// TIA Portal V20 export
TYPE "LKinCtrl_typePointParameter_reduced"
   STRUCT
      pathDynamics : "LKinCtrl_typePathDynamics";   // dynamics settings for single command
      orientationDirection : DInt := 3;   // 1: positive direction; 2: negative direction; 3: shortest distance
      bufferMode : DInt := 1;   // 1: standstill between commands, 2: blending with lower speed; 5: blending with higher speed
      transitionParameters : Array[1..5] of LReal;   // blending distance parameters
      dynamicAdaption : DInt := -1;   // <0.0: default TO setting used; 0: no dynamic adaption; 1: with variable limits; 2: with constant limits
   END_STRUCT;
   // transitionParameters[1] := -1.0;
END_TYPE
